FUNCTION_BLOCK FB_CylinderManualCtrl
VAR_INPUT
	bTrigger	: BOOL;
	Cylinder	: REFERENCE TO  FB_Cylinder; 
END_VAR
VAR_OUTPUT
END_VAR
VAR
	rTrig	:R_TRIG;
	fTrig	:F_TRIG;
END_VAR

rTrig(CLK:=bTrigger);
fTrig(CLK:=bTrigger);

IF rTrig.Q THEN
	Cylinder.M_Extend();
ELSIF fTrig.Q THEN
	Cylinder.M_Retract();
END_IF

END_FUNCTION_BLOCK

(* stored: Version 1.1.0.1, ProductVersion 3.1.4024.13
   POU FB_CylinderManualCtrl: Id {7c7c54ab-a9d0-49ee-8d3a-252702d8020d}, SpecialFunc None *)
